(* PLC project Office_Lighting, Actility iec61131 1.0.28, author Laurent Nicq *)
(* stored: creationDateTime 2013-03-20T17:09:43, version 1.0.0, modificationDateTime 2013-09-17T17:31:58 *)

(* Example for using the Sunset *)
PROGRAM POU_Astro_Using
  VAR_EXTERNAL
    GL_Astro_Status : DINT;  (* 0 if Astro started *)
    GL_Current_DateTime : DT;
    GL_SunSet_Time : DT;
    GL_SunRise_Time : DT;
  END_VAR
  VAR
    Information : STRING;
    astro_status : DINT := 0;
    delay_before : TIME := t#30s;
    time_remaining : TIME;  (* Helper for debug *)
    delay_after : TIME := t#45s;
  END_VAR
  VAR_EXTERNAL
    GL_Automatic_Light : BOOL;
  END_VAR
  VAR
    current_day : DINT;
  END_VAR

(* transition new_day *)
yday(GL_Current_DateTime)<> current_day;
/* check for a different day. Avoid dealing with 365-366 days case */
              
(* Need to wait for a new day before using a
SunSet value calculated by the Astro script *)
INITIAL_STEP Get_status:
  GET_STATUS_INLINE1(N);
END_STEP
ACTION GET_STATUS_INLINE1:
  astro_status:= GL_Astro_Status;
END_ACTION
TRANSITION FROM Get_status TO Display_Status
  := astro_status <>0;
END_TRANSITION
TRANSITION FROM Get_status TO Astro_OK
  := astro_status = 0;
END_TRANSITION
STEP Display_Status:
  DISPLAY_STATUS_INLINE2(P);
END_STEP
ACTION DISPLAY_STATUS_INLINE2:
  Information:='Astro is NOT RUNNING';
END_ACTION
TRANSITION FROM Display_Status TO Get_status
  := TRUE;
END_TRANSITION
STEP Astro_OK:
  ASTRO_OK_INLINE3(P);
  store_current_day(N);
  remaining(N);
END_STEP
ACTION ASTRO_OK_INLINE3:
  Information:='Astro is RUNNING';
END_ACTION
TRANSITION FROM Astro_OK TO Start_SunSet
  := GL_Current_DateTime > GL_SunSet_Time - delay_before;
END_TRANSITION
STEP Start_SunSet:
  START_SUNSET_INLINE4(P);
END_STEP
ACTION START_SUNSET_INLINE4:
  GL_Automatic_Light:=TRUE;
END_ACTION
TRANSITION FROM Start_SunSet TO Stop_SunSet
  := GL_Current_DateTime > (( GL_SunSet_Time - delay_before) + delay_after);
END_TRANSITION
STEP Stop_SunSet:
  STOP_SUNSET_INLINE5(P);
END_STEP
ACTION STOP_SUNSET_INLINE5:
  GL_Automatic_Light:=FALSE;
END_ACTION
TRANSITION FROM Stop_SunSet TO Get_status
  := new_day;
END_TRANSITION

ACTION store_current_day:
current_day:= yday(GL_Current_DateTime);
              
END_ACTION

ACTION remaining:
time_remaining:= SUB_DT_DT(GL_SunSet_Time , GL_Current_DateTime);
              
END_ACTION
END_PROGRAM

(* Distributes the Sunset Sunrise times *)
PROGRAM POU_Astro_Sun_Time
  VAR_EXTERNAL
    GL_SunSet_Time : DT;
    GL_SunRise_Time : DT;
    GL_Current_DateTime : DT;
    GL_Astro_Status : INT;
    GL_Lat : REAL;
    GL_Lon : REAL;
  END_VAR
  VAR
    Astro_Version : STRING := '1.1.2';
    current_day : DINT;
    Lat : REAL := 0;
    Lon : REAL := 0;
  END_VAR

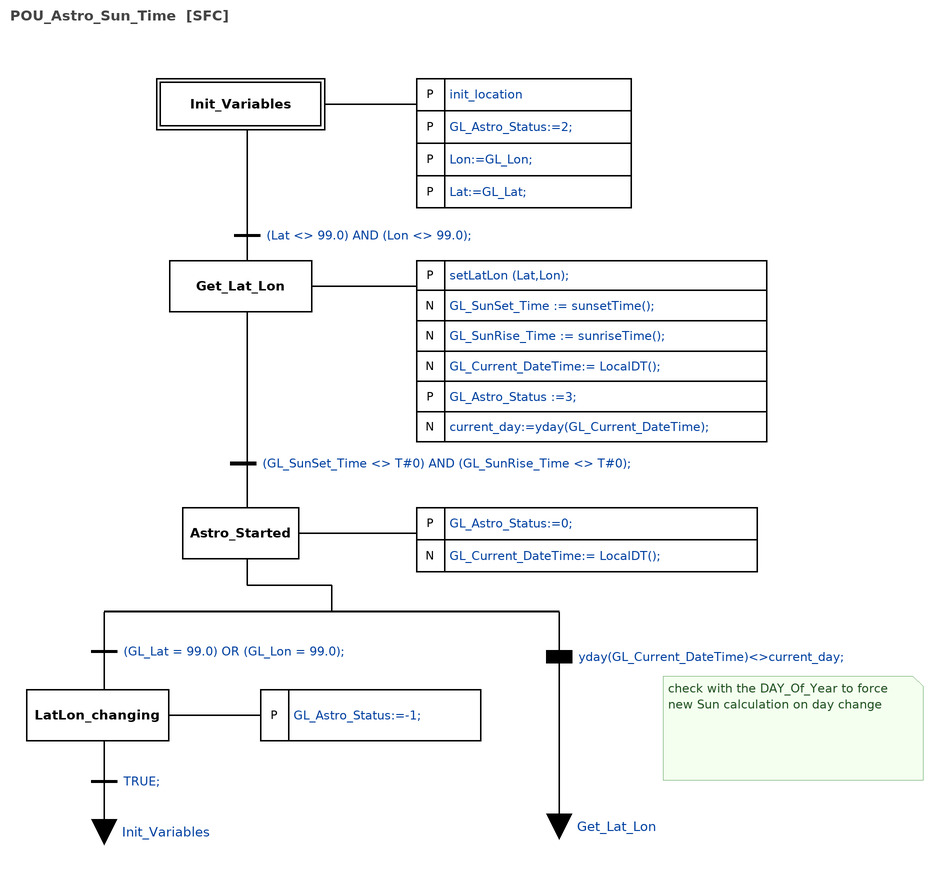
(* check with the DAY_Of_Year to force new Sun calculation on day change *)
INITIAL_STEP Init_Variables:
  init_location(P);
  INIT_VARIABLES_INLINE1(P);
  INIT_VARIABLES_INLINE2(P);
  INIT_VARIABLES_INLINE3(P);
END_STEP
ACTION INIT_VARIABLES_INLINE1:
  GL_Astro_Status:=2;
END_ACTION
ACTION INIT_VARIABLES_INLINE2:
  Lon:=GL_Lon;
END_ACTION
ACTION INIT_VARIABLES_INLINE3:
  Lat:=GL_Lat;
END_ACTION
TRANSITION FROM Init_Variables TO Get_Lat_Lon
  := (Lat <> 99.0) AND (Lon <> 99.0);
END_TRANSITION
STEP Get_Lat_Lon:
  GET_LAT_LON_INLINE4(P);
  GET_LAT_LON_INLINE5(N);
  GET_LAT_LON_INLINE6(N);
  GET_LAT_LON_INLINE7(N);
  GET_LAT_LON_INLINE8(P);
  GET_LAT_LON_INLINE9(N);
END_STEP
ACTION GET_LAT_LON_INLINE4:
  setLatLon (Lat,Lon);
END_ACTION
ACTION GET_LAT_LON_INLINE5:
  GL_SunSet_Time := sunsetTime();
END_ACTION
ACTION GET_LAT_LON_INLINE6:
  GL_SunRise_Time := sunriseTime();
END_ACTION
ACTION GET_LAT_LON_INLINE7:
  GL_Current_DateTime:= LocalDT();
END_ACTION
ACTION GET_LAT_LON_INLINE8:
  GL_Astro_Status :=3;
END_ACTION
ACTION GET_LAT_LON_INLINE9:
  current_day:=yday(GL_Current_DateTime);
END_ACTION
TRANSITION FROM Get_Lat_Lon TO Astro_Started
  := (GL_SunSet_Time <> T#0) AND (GL_SunRise_Time <> T#0);
END_TRANSITION
STEP Astro_Started:
  ASTRO_STARTED_INLINE10(P);
  ASTRO_STARTED_INLINE11(N);
END_STEP
ACTION ASTRO_STARTED_INLINE10:
  GL_Astro_Status:=0;
END_ACTION
ACTION ASTRO_STARTED_INLINE11:
  GL_Current_DateTime:= LocalDT();
END_ACTION
TRANSITION FROM Astro_Started TO LatLon_changing
  := (GL_Lat = 99.0) OR (GL_Lon = 99.0);
END_TRANSITION
TRANSITION FROM Astro_Started TO Get_Lat_Lon
  := yday(GL_Current_DateTime)<>current_day;
END_TRANSITION
STEP LatLon_changing:
  LATLON_CHANGING_INLINE12(P);
END_STEP
ACTION LATLON_CHANGING_INLINE12:
  GL_Astro_Status:=-1;
END_ACTION
TRANSITION FROM LatLon_changing TO Init_Variables
  := TRUE;
END_TRANSITION

ACTION init_location:
/* Lyon, France */
GL_Lat:=45.76404;
GL_Lon:=4.835659;
/* Narvik, Norway */
/* (no sunset in june and no sunrise in december) */
/* GL_Lat:=68.433; */
/* GL_Lon:=17.4167; */
              
END_ACTION
END_PROGRAM

(* Use Movemtent sensor as Presence sensor *)
PROGRAM Presence_detection
  VAR_EXTERNAL
    Move_Detected : BOOL;
    Move_Sensor : BOOL;
    Light_State1 : BOOL;
    Light_State2 : BOOL;
  END_VAR
  VAR
    Time_Stay_ON : TIME := t#20s;
    Running_time1 : TIME;
    Running_time2 : TIME;
    Pulse_Timer1 : TP;
    Pulse_Timer2 : TP;
    Rising_Edge : R_TRIG;
  END_VAR

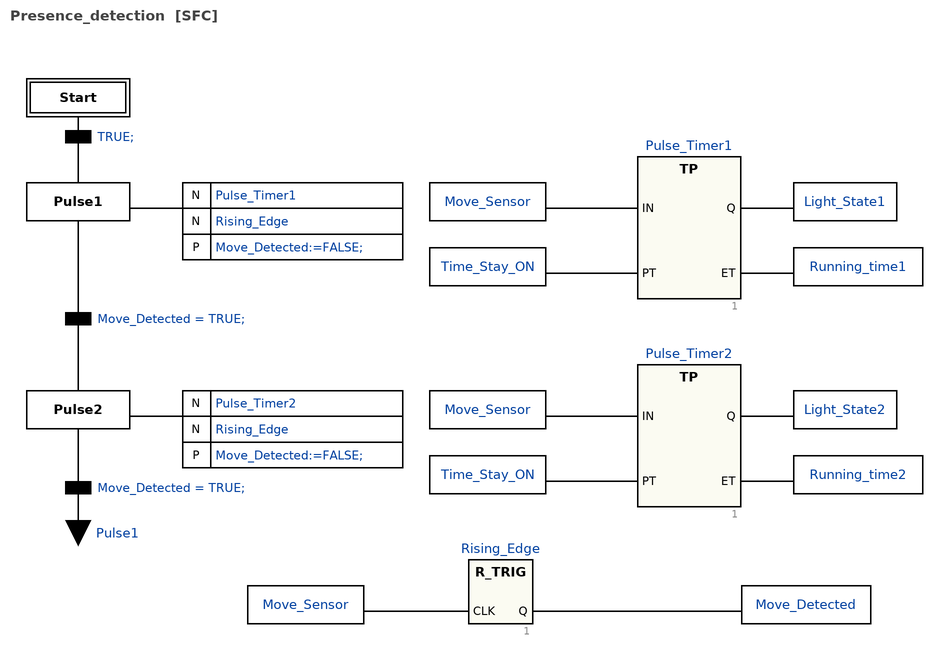
INITIAL_STEP Start:
  COMPUTE_FUNCTION_BLOCKS(S);
END_STEP
TRANSITION FROM Start TO Pulse1
  := TRUE;
END_TRANSITION
STEP Pulse1:
  Pulse_Timer1(N);
  Rising_Edge(N);
  PULSE1_INLINE1(P);
END_STEP
ACTION PULSE1_INLINE1:
  Move_Detected:=FALSE;
END_ACTION
TRANSITION FROM Pulse1 TO Pulse2
  := Move_Detected = TRUE;
END_TRANSITION
STEP Pulse2:
  Pulse_Timer2(N);
  Rising_Edge(N);
  PULSE2_INLINE2(P);
END_STEP
ACTION PULSE2_INLINE2:
  Move_Detected:=FALSE;
END_ACTION
TRANSITION FROM Pulse2 TO Pulse1
  := Move_Detected = TRUE;
END_TRANSITION
ACTION COMPUTE_FUNCTION_BLOCKS:  (* blocks drawn on the SFC sheet *)
  Pulse_Timer1(IN := Move_Sensor, PT := Time_Stay_ON);
  Pulse_Timer2(IN := Move_Sensor, PT := Time_Stay_ON);
  Rising_Edge(CLK := Move_Sensor);
  Light_State1 := Pulse_Timer1.Q;
  Running_time1 := Pulse_Timer1.ET;
  Light_State2 := Pulse_Timer2.Q;
  Running_time2 := Pulse_Timer2.ET;
  Move_Detected := Rising_Edge.Q;
END_ACTION
END_PROGRAM

(* Light Actuator Control *)
PROGRAM Light_control
  VAR_EXTERNAL
    Light_State1 : BOOL;
    Light_State2 : BOOL;
    Light_Actuator : BOOL;
    Move_Sensor : BOOL;
    Move_Detected : BOOL;
    GL_Automatic_Light : BOOL;
  END_VAR
  VAR  (* added by the conversion: wires and edge detectors of the diagram *)
    _OR2_OUT : BOOL;
    _AND1_OUT : BOOL;
  END_VAR

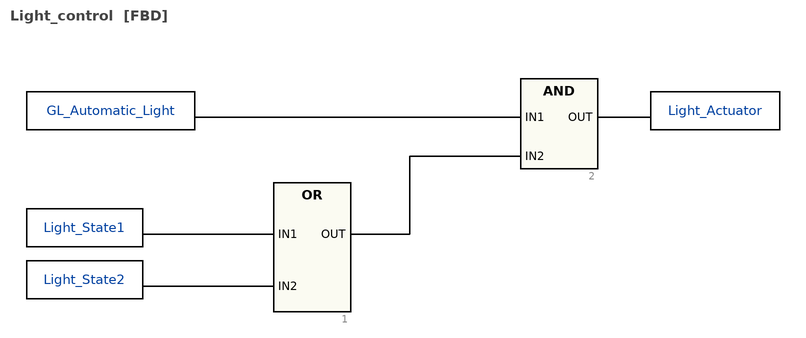
(* FBD diagram, written out as Structured Text *)
_OR2_OUT := Light_State1 OR Light_State2;
_AND1_OUT := GL_Automatic_Light AND _OR2_OUT;
Light_Actuator := _AND1_OUT;
END_PROGRAM

CONFIGURATION Astro_test
  RESOURCE Resource_main ON PLC
    VAR_GLOBAL
      GL_Automatic_Light : BOOL;  (* TRUE: automatic lighting at Night *)
      Light_Actuator : BOOL;
      Light_State1 : BOOL;  (* For first TP block *)
      Light_State2 : BOOL;  (* For second TP block *)
      Move_Sensor : BOOL := FALSE;  (* Movement detector *)
      Move_Detected : BOOL := FALSE;  (* Movement detected *)
      GL_SunSet_Time : DT := T#0;
      GL_SunRise_Time : DT := T#0;
      GL_Current_DateTime : DT;
      GL_Astro_Status : DINT := -1;  (* -1 means Stopped *)
      GL_Lat : REAL := -99.0;  (* -99.0 means not initialized *)
      GL_Lon : REAL := -99.0;  (* -99.0 means not initialized *)
    END_VAR
    TASK task_slow(INTERVAL := T#5s0ms, PRIORITY := 0);
    TASK task_fast(INTERVAL := T#1s0ms, PRIORITY := 0);
    PROGRAM Instance_Astro_calc WITH task_slow : POU_Astro_Sun_Time;
    PROGRAM Instance_Astro_use WITH task_fast : POU_Astro_Using;
    PROGRAM Presence WITH task_fast : Presence_detection;
    PROGRAM Lighting WITH task_fast : Light_control;
  END_RESOURCE
END_CONFIGURATION
